TYPE ST_HMI_InputSource : 
STRUCT
	nID: DINT;
	sDisplayName: WSTRING(80);
	
	sStreamSystemID: GUID;
	sTopic: STRING(255);
	
	eSourceType: E_SourceType;;
	eState: E_DataSourceState;;
	dtTimestamp: DCTIMESTRUCT;
	
	stHist: ST_HMI_DataSourceHist;
END_STRUCT
END_TYPE

(* stored: DUT ST_HMI_InputSource: Id c4433802-91ac-4f04-9c02-9654fcf40f2c *)
